INTERFACE I_Pause

METHOD Pause
VAR_INPUT
	bPause 		:  BOOL; // Pause Timer (TRUE), Only Pauses if IN := TRUE.
END_VAR
END_METHOD

END_INTERFACE

(* stored: Version 1.1.0.1, ProductVersion 3.1.4024.12
   Itf I_Pause: Id {29925558-0fa7-4c17-b625-aec698ef5741}
   Method Pause: Id {bb623033-c04f-44ec-b93a-dec8f1de4c22} *)
